# EPICS substitutions: apps/ftIntlkApp/Db/ftcIntlk.substitutions
file "db/ftcIntlk_hvQstat.db" {
pattern {P Q}
    {B_DET_FTC_ 1}
    {B_DET_FTC_ 2}
    {B_DET_FTC_ 3}
    {B_DET_FTC_ 4}
}
file "db/ftcIntlk_lvQ2.db" {
pattern {P Q1 Q2}
    {B_DET_FTC_ 1 4}
    {B_DET_FTC_ 2 3}
}
